LIN {X 0,Y 29.595,Z 545.275,A -85,B 0,C 180,E1 -30358.352,E2 -30358.352} C_VEL
LIN {X 0,Y 37.281,Z 542.804,A -85,B 0,C 180,E1 -30378.939,E2 -30378.939} C_VEL
LIN {X 0,Y 45.185,Z 539.847,A -85,B 0,C 180,E1 -30388.806,E2 -30388.806} C_VEL
LIN {X 0,Y 53.99,Z 535.853,A -85,B 0,C 180,E1 -30395.667,E2 -30395.667} C_VEL
LIN {X 0,Y 63.603,Z 530.542,A -85,B 0,C 180,E1 -30400.777,E2 -30400.777} C_VEL
LIN {X 0,Y 68.114,Z 527.764,A -85,B 0,C 180,E1 -30402.626,E2 -30402.626} C_VEL
LIN {X 0,Y 69.579,Z 526.593,A -85,B 0,C 180,E1 -30403.646,E2 -30403.646} C_VEL
LIN {X 0,Y 71.55,Z 524.834,A -85,B 0,C 180,E1 -30405.785,E2 -30405.785} C_VEL
LIN {X 0,Y 72.682,Z 523.453,A -85,B 0,C 180,E1 -30408.846,E2 -30408.846} C_VEL
LIN {X 0,Y 73.708,Z 521.841,A -85,B 0,C 180,E1 -30414.526,E2 -30414.526} C_VEL
LIN {X 0,Y 74.494,Z 520.765,A -85,B 0,C 180,E1 -30419.997,E2 -30419.997} C_VEL
LIN {X 0,Y 73.406,Z 521.71,A -85,B 0,C 180,E1 -30426.874,E2 -30426.874} C_VEL
LIN {X 0,Y 72.504,Z 523.18,A -85,B 0,C 180,E1 -30434.237,E2 -30434.237} C_VEL
LIN {X 0,Y 72.199,Z 523.884,A -85,B 0,C 180,E1 -30436.976,E2 -30436.976} C_VEL
LIN {X 0,Y 70.741,Z 526.379,A -85,B 0,C 180,E1 -30443.412,E2 -30443.412} C_VEL
LIN {X 0,Y 69.633,Z 527.972,A -85,B 0,C 180,E1 -30447.263,E2 -30447.263} C_VEL
LIN {X 0,Y 67.359,Z 530.893,A -85,B 0,C 180,E1 -30453.419,E2 -30453.419} C_VEL
LIN {X 0,Y 63.449,Z 535.475,A -85,B 0,C 180,E1 -30464.224,E2 -30464.224} C_VEL
LIN {X 0,Y 61.857,Z 538.776,A -85,B 0,C 180,E1 -30475.385,E2 -30475.385} C_VEL
LIN {X 0,Y 62.441,Z 540.641,A -85,B 0,C 180,E1 -30484.207,E2 -30484.207} C_VEL
LIN {X 0,Y 67.081,Z 542.547,A -85,B 0,C 180,E1 -30497.906,E2 -30497.906} C_VEL
LIN {X 0,Y 71.274,Z 542.971,A -85,B 0,C 180,E1 -30504.342,E2 -30504.342} C_VEL
LIN {X 0,Y 76.407,Z 542.961,A -85,B 0,C 180,E1 -30510.001,E2 -30510.001} C_VEL
LIN {X 0,Y 70.708,Z 542.926,A -85,B 0,C 180,E1 -30516.34,E2 -30516.34} C_VEL
LIN {X 0,Y 65.558,Z 542.209,A -85,B 0,C 180,E1 -30525.255,E2 -30525.255} C_VEL
LIN {X 0,Y 62.285,Z 540.421,A -85,B 0,C 180,E1 -30536.831,E2 -30536.831} C_VEL
LIN {X 0,Y 61.937,Z 538.036,A -85,B 0,C 180,E1 -30547.417,E2 -30547.417} C_VEL
LIN {X 0,Y 64.403,Z 534.161,A -85,B 0,C 180,E1 -30559.104,E2 -30559.104} C_VEL
LIN {X 0,Y 67.352,Z 530.892,A -85,B 0,C 180,E1 -30566.594,E2 -30566.594} C_VEL
LIN {X 0,Y 69.62,Z 527.97,A -85,B 0,C 180,E1 -30572.767,E2 -30572.767} C_VEL
LIN {X 0,Y 70.694,Z 526.411,A -85,B 0,C 180,E1 -30576.572,E2 -30576.572} C_VEL
LIN {X 0,Y 72.192,Z 523.889,A -85,B 0,C 180,E1 -30583.022,E2 -30583.022} C_VEL
LIN {X 0,Y 72.928,Z 522.452,A -85,B 0,C 180,E1 -30588.89,E2 -30588.89} C_VEL
LIN {X 0,Y 73.661,Z 521.458,A -85,B 0,C 180,E1 -30594.528,E2 -30594.528} C_VEL
LIN {X 0,Y 74.463,Z 520.789,A -85,B 0,C 180,E1 -30600.003,E2 -30600.003} C_VEL
LIN {X 0,Y 73.535,Z 522.043,A -85,B 0,C 180,E1 -30606.153,E2 -30606.153} C_VEL
LIN {X 0,Y 72.336,Z 523.174,A -85,B 0,C 180,E1 -30608.285,E2 -30608.285} C_VEL
LIN {X 0,Y 69.882,Z 525.092,A -85,B 0,C 180,E1 -30610.206,E2 -30610.206} C_VEL
LIN {X 0,Y 67.39,Z 526.857,A -85,B 0,C 180,E1 -30611.352,E2 -30611.352} C_VEL
LIN {X 0,Y 57.594,Z 532.628,A -85,B 0,C 180,E1 -30614.394,E2 -30614.394} C_VEL
LIN {X 0,Y 48.232,Z 537.171,A -85,B 0,C 180,E1 -30618.71,E2 -30618.71} C_VEL
LIN {X 0,Y 38.881,Z 540.786,A -85,B 0,C 180,E1 -30625.336,E2 -30625.336} C_VEL
LIN {X 0,Y 33.037,Z 542.591,A -85,B 0,C 180,E1 -30631.685,E2 -30631.685} C_VEL
LIN {X 0,Y 23.563,Z 545.062,A -85,B 0,C 180,E1 -30653.374,E2 -30653.374} C_VEL
LIN {X 0,Y 20.769,Z 545.664,A -85,B 0,C 180,E1 -30670.217,E2 -30670.217} C_VEL
LIN {X 0,Y 20.025,Z 545.83,A -85,B 0,C 180,E1 -30689.996,E2 -30689.996} C_VEL
LIN {X 0,Y 20.768,Z 545.664,A -85,B 0,C 180,E1 -30709.775,E2 -30709.775} C_VEL
LIN {X 0,Y 23.561,Z 545.062,A -85,B 0,C 180,E1 -30726.62,E2 -30726.62} C_VEL
LIN {X 0,Y 33.035,Z 542.592,A -85,B 0,C 180,E1 -30748.313,E2 -30748.313} C_VEL
LIN {X 0,Y 41.939,Z 539.635,A -85,B 0,C 180,E1 -30757.165,E2 -30757.165} C_VEL
LIN {X 0,Y 51.468,Z 535.641,A -85,B 0,C 180,E1 -30762.905,E2 -30762.905} C_VEL
LIN {X 0,Y 61.319,Z 530.507,A -85,B 0,C 180,E1 -30766.938,E2 -30766.938} C_VEL
LIN {X 0,Y 64.658,Z 528.588,A -85,B 0,C 180,E1 -30768.017,E2 -30768.017} C_VEL
LIN {X 0,Y 66.911,Z 526.732,A -85,B 0,C 180,E1 -30771.207,E2 -30771.207} C_VEL
LIN {X 0,Y 67.428,Z 526.025,A -85,B 0,C 180,E1 -30774.014,E2 -30774.014} C_VEL
LIN {X 0,Y 68.512,Z 524.866,A -85,B 0,C 180,E1 -30779.997,E2 -30779.997} C_VEL
LIN {X 0,Y 67.504,Z 525.562,A -85,B 0,C 180,E1 -30786.094,E2 -30786.094} C_VEL
LIN {X 0,Y 66.682,Z 526.625,A -85,B 0,C 180,E1 -30792.165,E2 -30792.165} C_VEL
LIN {X 0,Y 65.975,Z 527.63,A -85,B 0,C 180,E1 -30796.526,E2 -30796.526} C_VEL
LIN {X 0,Y 64.335,Z 529.517,A -85,B 0,C 180,E1 -30802.475,E2 -30802.475} C_VEL
LIN {X 0,Y 62.896,Z 531.158,A -85,B 0,C 180,E1 -30806.635,E2 -30806.635} C_VEL
LIN {X 0,Y 61.261,Z 532.718,A -85,B 0,C 180,E1 -30810.64,E2 -30810.64} C_VEL
LIN {X 0,Y 56.854,Z 536.807,A -85,B 0,C 180,E1 -30822.128,E2 -30822.128} C_VEL
LIN {X 0,Y 55.221,Z 539.024,A -85,B 0,C 180,E1 -30830.482,E2 -30830.482} C_VEL
LIN {X 0,Y 55.213,Z 541.318,A -85,B 0,C 180,E1 -30842.993,E2 -30842.993} C_VEL
LIN {X 0,Y 58.568,Z 542.807,A -85,B 0,C 180,E1 -30856.116,E2 -30856.116} C_VEL
LIN {X 0,Y 63.481,Z 543.319,A -85,B 0,C 180,E1 -30865.084,E2 -30865.084} C_VEL
LIN {X 0,Y 67.405,Z 543.228,A -85,B 0,C 180,E1 -30870.001,E2 -30870.001} C_VEL
LIN {X 0,Y 62.439,Z 543.236,A -85,B 0,C 180,E1 -30876.464,E2 -30876.464} C_VEL
LIN {X 0,Y 58.183,Z 542.744,A -85,B 0,C 180,E1 -30884.925,E2 -30884.925} C_VEL
LIN {X 0,Y 54.911,Z 540.671,A -85,B 0,C 180,E1 -30900.796,E2 -30900.796} C_VEL
LIN {X 0,Y 55.817,Z 537.952,A -85,B 0,C 180,E1 -30913.825,E2 -30913.825} C_VEL
LIN {X 0,Y 59.648,Z 534.186,A -85,B 0,C 180,E1 -30925.566,E2 -30925.566} C_VEL
LIN {X 0,Y 61.25,Z 532.717,A -85,B 0,C 180,E1 -30929.382,E2 -30929.382} C_VEL
LIN {X 0,Y 62.895,Z 531.138,A -85,B 0,C 180,E1 -30933.455,E2 -30933.455} C_VEL
LIN {X 0,Y 64.302,Z 529.536,A -85,B 0,C 180,E1 -30937.513,E2 -30937.513} C_VEL
LIN {X 0,Y 65.967,Z 527.63,A -85,B 0,C 180,E1 -30943.508,E2 -30943.508} C_VEL
LIN {X 0,Y 66.69,Z 526.619,A -85,B 0,C 180,E1 -30947.836,E2 -30947.836} C_VEL
LIN {X 0,Y 67.533,Z 525.536,A -85,B 0,C 180,E1 -30954.03,E2 -30954.03} C_VEL
LIN {X 0,Y 68.475,Z 524.89,A -85,B 0,C 180,E1 -30960.003,E2 -30960.003} C_VEL
LIN {X 0,Y 67.404,Z 526.04,A -85,B 0,C 180,E1 -30965.988,E2 -30965.988} C_VEL
LIN {X 0,Y 66.816,Z 526.795,A -85,B 0,C 180,E1 -30968.807,E2 -30968.807} C_VEL
LIN {X 0,Y 64.662,Z 528.587,A -85,B 0,C 180,E1 -30971.986,E2 -30971.986} C_VEL
LIN {X 0,Y 57.594,Z 532.628,A -85,B 0,C 180,E1 -30974.394,E2 -30974.394} C_VEL
LIN {X 0,Y 52.388,Z 535.105,A -85,B 0,C 180,E1 -30975.853,E2 -30975.853} C_VEL
LIN {X 0,Y 46.882,Z 537.38,A -85,B 0,C 180,E1 -30976.499,E2 -30976.499} C_VEL
LIN {X 0,Y 35.537,Z 540.932,A -85,B 0,C 180,E1 -30977.575,E2 -30977.575} C_VEL
LIN {X 0,Y 29.088,Z 542.618,A -85,B 0,C 180,E1 -30980.837,E2 -30980.837} C_VEL
LIN {X 0,Y 28.223,Z 542.755,A -85,B 0,C 180,E1 -30981.7,E2 -30981.7} C_VEL
LIN {X 0,Y 18.344,Z 544.85,A -85,B 0,C 180,E1 -30999.978,E2 -30999.978} C_VEL
LIN {X 0,Y 14.273,Z 545.452,A -85,B 0,C 180,E1 -31020.494,E2 -31020.494} C_VEL
LIN {X 0,Y 12.932,Z 545.619,A -85,B 0,C 180,E1 -31049.993,E2 -31049.993} C_VEL
LIN {X 0,Y 14.271,Z 545.452,A -85,B 0,C 180,E1 -31079.495,E2 -31079.495} C_VEL
LIN {X 0,Y 18.342,Z 544.85,A -85,B 0,C 180,E1 -31100.016,E2 -31100.016} C_VEL
LIN {X 0,Y 29.909,Z 542.38,A -85,B 0,C 180,E1 -31120.024,E2 -31120.024} C_VEL
LIN {X 0,Y 39.72,Z 539.422,A -85,B 0,C 180,E1 -31126.685,E2 -31126.685} C_VEL
LIN {X 0,Y 49.842,Z 535.429,A -85,B 0,C 180,E1 -31130.75,E2 -31130.75} C_VEL
LIN {X 0,Y 60.111,Z 530.295,A -85,B 0,C 180,E1 -31133.565,E2 -31133.565} C_VEL
LIN {X 0,Y 61.605,Z 529.239,A -85,B 0,C 180,E1 -31136.726,E2 -31136.726} C_VEL
LIN {X 0,Y 62.267,Z 528.721,A -85,B 0,C 180,E1 -31139.996,E2 -31139.996} C_VEL
LIN {X 0,Y 61.158,Z 529.332,A -85,B 0,C 180,E1 -31146.595,E2 -31146.595} C_VEL
LIN {X 0,Y 60.017,Z 530.426,A -85,B 0,C 180,E1 -31153.541,E2 -31153.541} C_VEL
LIN {X 0,Y 58.992,Z 531.466,A -85,B 0,C 180,E1 -31157.629,E2 -31157.629} C_VEL
LIN {X 0,Y 57.693,Z 532.582,A -85,B 0,C 180,E1 -31161.431,E2 -31161.431} C_VEL
LIN {X 0,Y 55.312,Z 534.438,A -85,B 0,C 180,E1 -31167.203,E2 -31167.203} C_VEL
LIN {X 0,Y 51.732,Z 537.05,A -85,B 0,C 180,E1 -31175.405,E2 -31175.405} C_VEL
LIN {X 0,Y 48.796,Z 539.572,A -85,B 0,C 180,E1 -31186.059,E2 -31186.059} C_VEL
LIN {X 0,Y 48.243,Z 542.159,A -85,B 0,C 180,E1 -31204.087,E2 -31204.087} C_VEL
LIN {X 0,Y 50.802,Z 543.149,A -85,B 0,C 180,E1 -31215.538,E2 -31215.538} C_VEL
LIN {X 0,Y 56.3,Z 543.561,A -85,B 0,C 180,E1 -31226.94,E2 -31226.94} C_VEL
LIN {X 0,Y 58.461,Z 543.495,A -85,B 0,C 180,E1 -31230.001,E2 -31230.001} C_VEL
LIN {X 0,Y 53.721,Z 543.497,A -85,B 0,C 180,E1 -31237.519,E2 -31237.519} C_VEL
LIN {X 0,Y 50.276,Z 543.063,A -85,B 0,C 180,E1 -31246.237,E2 -31246.237} C_VEL
LIN {X 0,Y 48.02,Z 541.878,A -85,B 0,C 180,E1 -31258.592,E2 -31258.592} C_VEL
LIN {X 0,Y 49.079,Z 539.271,A -85,B 0,C 180,E1 -31275.726,E2 -31275.726} C_VEL
LIN {X 0,Y 53.19,Z 536.073,A -85,B 0,C 180,E1 -31288.099,E2 -31288.099} C_VEL
LIN {X 0,Y 55.302,Z 534.438,A -85,B 0,C 180,E1 -31292.823,E2 -31292.823} C_VEL
LIN {X 0,Y 57.64,Z 532.607,A -85,B 0,C 180,E1 -31298.548,E2 -31298.548} C_VEL
LIN {X 0,Y 58.984,Z 531.465,A -85,B 0,C 180,E1 -31302.407,E2 -31302.407} C_VEL
LIN {X 0,Y 60.014,Z 530.428,A -85,B 0,C 180,E1 -31306.459,E2 -31306.459} C_VEL
LIN {X 0,Y 61.163,Z 529.33,A -85,B 0,C 180,E1 -31313.406,E2 -31313.406} C_VEL
LIN {X 0,Y 62.253,Z 528.729,A -85,B 0,C 180,E1 -31320.004,E2 -31320.004} C_VEL
LIN {X 0,Y 61.578,Z 529.254,A -85,B 0,C 180,E1 -31323.275,E2 -31323.275} C_VEL
LIN {X 0,Y 60.113,Z 530.294,A -85,B 0,C 180,E1 -31326.429,E2 -31326.429} C_VEL
LIN {X 0,Y 49.845,Z 535.428,A -85,B 0,C 180,E1 -31329.253,E2 -31329.253} C_VEL
LIN {X 0,Y 39.723,Z 539.421,A -85,B 0,C 180,E1 -31333.316,E2 -31333.316} C_VEL
LIN {X 0,Y 29.912,Z 542.379,A -85,B 0,C 180,E1 -31339.974,E2 -31339.974} C_VEL
LIN {X 0,Y 28.223,Z 542.755,A -85,B 0,C 180,E1 -31341.7,E2 -31341.7} C_VEL
LIN {X 0,Y 22.938,Z 543.892,A -85,B 0,C 180,E1 -31347.166,E2 -31347.166} C_VEL
LIN {X 0,Y 17.452,Z 544.74,A -85,B 0,C 180,E1 -31353.279,E2 -31353.279} C_VEL
LIN {X 0,Y 7.362,Z 545.435,A -85,B 0,C 180,E1 -31386.239,E2 -31386.239} C_VEL
LIN {X 0,Y 7.357,Z 545.291,A -85,B 0,C 180,E1 -31452.017,E2 -31452.017} C_VEL
LIN {X 0,Y 14.81,Z 544.638,A -85,B 0,C 180,E1 -31481.617,E2 -31481.617} C_VEL
LIN {X 0,Y 28.279,Z 542.167,A -85,B 0,C 180,E1 -31493.727,E2 -31493.727} C_VEL
LIN {X 0,Y 38.705,Z 539.21,A -85,B 0,C 180,E1 -31497.007,E2 -31497.007} C_VEL
LIN {X 0,Y 49.201,Z 535.216,A -85,B 0,C 180,E1 -31498.992,E2 -31498.992} C_VEL
LIN {X 0,Y 55.815,Z 532.215,A -85,B 0,C 180,E1 -31499.996,E2 -31499.996} C_VEL
LIN {X 0,Y 54.509,Z 532.847,A -85,B 0,C 180,E1 -31507.404,E2 -31507.404} C_VEL
LIN {X 0,Y 52.661,Z 534.088,A -85,B 0,C 180,E1 -31515.476,E2 -31515.476} C_VEL
LIN {X 0,Y 51.739,Z 534.714,A -85,B 0,C 180,E1 -31518.047,E2 -31518.047} C_VEL
LIN {X 0,Y 49.656,Z 536.09,A -85,B 0,C 180,E1 -31522.702,E2 -31522.702} C_VEL
LIN {X 0,Y 43.786,Z 539.514,A -85,B 0,C 180,E1 -31536.631,E2 -31536.631} C_VEL
LIN {X 0,Y 41.503,Z 541.167,A -85,B 0,C 180,E1 -31547.367,E2 -31547.367} C_VEL
LIN {X 0,Y 42.116,Z 543.318,A -85,B 0,C 180,E1 -31570.506,E2 -31570.506} C_VEL
LIN {X 0,Y 45.091,Z 543.757,A -85,B 0,C 180,E1 -31581.035,E2 -31581.035} C_VEL
LIN {X 0,Y 49.616,Z 543.758,A -85,B 0,C 180,E1 -31590.002,E2 -31590.002} C_VEL
LIN {X 0,Y 43.443,Z 543.542,A -85,B 0,C 180,E1 -31603.936,E2 -31603.936} C_VEL
LIN {X 0,Y 40.872,Z 542.408,A -85,B 0,C 180,E1 -31621.057,E2 -31621.057} C_VEL
LIN {X 0,Y 42.45,Z 540.3,A -85,B 0,C 180,E1 -31638.536,E2 -31638.536} C_VEL
LIN {X 0,Y 48.026,Z 536.976,A -85,B 0,C 180,E1 -31653.965,E2 -31653.965} C_VEL
LIN {X 0,Y 49.641,Z 536.094,A -85,B 0,C 180,E1 -31657.316,E2 -31657.316} C_VEL
LIN {X 0,Y 51.71,Z 534.715,A -85,B 0,C 180,E1 -31662.064,E2 -31662.064} C_VEL
LIN {X 0,Y 52.615,Z 534.109,A -85,B 0,C 180,E1 -31664.51,E2 -31664.51} C_VEL
LIN {X 0,Y 54.511,Z 532.845,A -85,B 0,C 180,E1 -31672.597,E2 -31672.597} C_VEL
LIN {X 0,Y 55.806,Z 532.22,A -85,B 0,C 180,E1 -31680.004,E2 -31680.004} C_VEL
LIN {X 0,Y 45.7,Z 536.747,A -85,B 0,C 180,E1 -31681.554,E2 -31681.554} C_VEL
LIN {X 0,Y 35.222,Z 540.362,A -85,B 0,C 180,E1 -31683.893,E2 -31683.893} C_VEL
LIN {X 0,Y 25.646,Z 542.703,A -85,B 0,C 180,E1 -31687.603,E2 -31687.603} C_VEL
LIN {X 0,Y 14.813,Z 544.638,A -85,B 0,C 180,E1 -31698.38,E2 -31698.38} C_VEL
LIN {X 0,Y 8.81,Z 545.24,A -85,B 0,C 180,E1 -31717.075,E2 -31717.075} C_VEL
LIN {X 0,Y 5.826,Z 545.408,A -85,B 0,C 180,E1 -31769.985,E2 -31769.985} C_VEL
LIN {X 0,Y 7.357,Z 545.291,A -85,B 0,C 180,E1 -31812.017,E2 -31812.017} C_VEL
LIN {X 0,Y 10.044,Z 545.109,A -85,B 0,C 180,E1 -31831.192,E2 -31831.192} C_VEL
LIN {X 0,Y 16.341,Z 544.329,A -85,B 0,C 180,E1 -31852.358,E2 -31852.358} C_VEL
LIN {X 0,Y 27.025,Z 542.304,A -85,B 0,C 180,E1 -31865.805,E2 -31865.805} C_VEL
LIN {X 0,Y 32.715,Z 540.862,A -85,B 0,C 180,E1 -31867.68,E2 -31867.68} C_VEL
LIN {X 0,Y 34.634,Z 540.361,A -85,B 0,C 180,E1 -31867.71,E2 -31867.71} C_VEL
LIN {X 0,Y 42.529,Z 537.777,A -85,B 0,C 180,E1 -31867.489,E2 -31867.489} C_VEL
LIN {X 0,Y 47.334,Z 536.029,A -85,B 0,C 180,E1 -31868.534,E2 -31868.534} C_VEL
LIN {X 0,Y 44.177,Z 537.55,A -85,B 0,C 180,E1 -31877.355,E2 -31877.355} C_VEL
LIN {X 0,Y 39.462,Z 539.757,A -85,B 0,C 180,E1 -31887.073,E2 -31887.073} C_VEL
LIN {X 0,Y 35.838,Z 541.414,A -85,B 0,C 180,E1 -31898.338,E2 -31898.338} C_VEL
LIN {X 0,Y 34.257,Z 543.57,A -85,B 0,C 180,E1 -31925.779,E2 -31925.779} C_VEL
LIN {X 0,Y 36.638,Z 544.012,A -85,B 0,C 180,E1 -31938.943,E2 -31938.943} C_VEL
LIN {X 0,Y 40.886,Z 544.018,A -85,B 0,C 180,E1 -31950.002,E2 -31950.002} C_VEL
LIN {X 0,Y 36.079,Z 543.94,A -85,B 0,C 180,E1 -31963.127,E2 -31963.127} C_VEL
LIN {X 0,Y 33.821,Z 542.994,A -85,B 0,C 180,E1 -31983.789,E2 -31983.789} C_VEL
LIN {X 0,Y 36.567,Z 540.999,A -85,B 0,C 180,E1 -32004.797,E2 -32004.797} C_VEL
LIN {X 0,Y 39.444,Z 539.758,A -85,B 0,C 180,E1 -32012.989,E2 -32012.989} C_VEL
LIN {X 0,Y 44.168,Z 537.55,A -85,B 0,C 180,E1 -32022.697,E2 -32022.697} C_VEL
LIN {X 0,Y 47.3,Z 536.044,A -85,B 0,C 180,E1 -32031.46,E2 -32031.46} C_VEL
LIN {X 0,Y 42.531,Z 537.776,A -85,B 0,C 180,E1 -32032.514,E2 -32032.514} C_VEL
LIN {X 0,Y 35.457,Z 540.15,A -85,B 0,C 180,E1 -32032.34,E2 -32032.34} C_VEL
LIN {X 0,Y 28.401,Z 541.955,A -85,B 0,C 180,E1 -32031.84,E2 -32031.84} C_VEL
LIN {X 0,Y 14.27,Z 544.426,A -85,B 0,C 180,E1 -32030.088,E2 -32030.088} C_VEL
LIN {X 0,Y 7.253,Z 545.029,A -85,B 0,C 180,E1 -32025.723,E2 -32025.723} C_VEL
LIN {X 0,Y 1.286,Z 545.196,A -85,B 0,C 180,E1 -31950.068,E2 -31950.068} C_VEL
LIN {X 0,Y 7.25,Z 545.029,A -85,B 0,C 180,E1 -31874.283,E2 -31874.283} C_VEL
LIN {X 0,Y 14.267,Z 544.426,A -85,B 0,C 180,E1 -31869.914,E2 -31869.914} C_VEL
LIN {X 0,Y 28.398,Z 541.955,A -85,B 0,C 180,E1 -31868.162,E2 -31868.162} C_VEL
LIN {X 0,Y 34.634,Z 540.361,A -85,B 0,C 180,E1 -31867.71,E2 -31867.71} C_VEL
LIN {X 0,Y 35.253,Z 540.211,A -85,B 0,C 180,E1 -31868.775,E2 -31868.775} C_VEL
LIN {X 0,Y 35.21,Z 540.264,A -85,B 0,C 180,E1 -31872.001,E2 -31872.001} C_VEL
LIN {X 0,Y 33.985,Z 540.688,A -85,B 0,C 180,E1 -31877.327,E2 -31877.327} C_VEL
LIN {X 0,Y 29.844,Z 542.226,A -85,B 0,C 180,E1 -31890.972,E2 -31890.972} C_VEL
LIN {X 0,Y 27.416,Z 543.169,A -85,B 0,C 180,E1 -31905.259,E2 -31905.259} C_VEL
LIN {X 0,Y 28.304,Z 544.266,A -85,B 0,C 180,E1 -31935.626,E2 -31935.626} C_VEL
LIN {X 0,Y 32.248,Z 544.275,A -85,B 0,C 180,E1 -31950.003,E2 -31950.003} C_VEL
LIN {X 0,Y 28.306,Z 544.266,A -85,B 0,C 180,E1 -31964.379,E2 -31964.379} C_VEL
LIN {X 0,Y 26.882,Z 543.558,A -85,B 0,C 180,E1 -31988.355,E2 -31988.355} C_VEL
LIN {X 0,Y 32.945,Z 541.106,A -85,B 0,C 180,E1 -32017.598,E2 -32017.598} C_VEL
LIN {X 0,Y 30.242,Z 541.743,A -85,B 0,C 180,E1 -32018.371,E2 -32018.371} C_VEL
LIN {X 0,Y 17.023,Z 544.213,A -85,B 0,C 180,E1 -32005.666,E2 -32005.666} C_VEL
LIN {X 0,Y 11.353,Z 544.817,A -85,B 0,C 180,E1 -31988.255,E2 -31988.255} C_VEL
LIN {X 0,Y 8.384,Z 544.985,A -85,B 0,C 180,E1 -31950.01,E2 -31950.01} C_VEL
LIN {X 0,Y 11.351,Z 544.817,A -85,B 0,C 180,E1 -31911.757,E2 -31911.757} C_VEL
LIN {X 0,Y 17.021,Z 544.214,A -85,B 0,C 180,E1 -31894.34,E2 -31894.34} C_VEL
LIN {X 0,Y 30.24,Z 541.744,A -85,B 0,C 180,E1 -31881.632,E2 -31881.632} C_VEL
LIN {X 0,Y 32.979,Z 541.099,A -85,B 0,C 180,E1 -31882.44,E2 -31882.44} C_VEL
LIN {X 0,Y 27.416,Z 543.169,A -85,B 0,C 180,E1 -31905.259,E2 -31905.259} C_VEL
LIN {X 0,Y 26.068,Z 543.59,A -85,B 0,C 180,E1 -31910.071,E2 -31910.071} C_VEL
LIN {X 0,Y 20.556,Z 544.355,A -85,B 0,C 180,E1 -31922.928,E2 -31922.928} C_VEL
LIN {X 0,Y 20.177,Z 544.509,A -85,B 0,C 180,E1 -31929.171,E2 -31929.171} C_VEL
LIN {X 0,Y 23.622,Z 544.531,A -85,B 0,C 180,E1 -31950.004,E2 -31950.004} C_VEL
LIN {X 0,Y 19.788,Z 544.377,A -85,B 0,C 180,E1 -31977.889,E2 -31977.889} C_VEL
LIN {X 0,Y 17.506,Z 544.605,A -85,B 0,C 180,E1 -31973.675,E2 -31973.675} C_VEL
LIN {X 0,Y 15.473,Z 544.774,A -85,B 0,C 180,E1 -31950.006,E2 -31950.006} C_VEL
LIN {X 0,Y 17.504,Z 544.605,A -85,B 0,C 180,E1 -31926.334,E2 -31926.334} C_VEL
LIN {X 0,Y 19.795,Z 544.376,A -85,B 0,C 180,E1 -31922.094,E2 -31922.094} C_VEL
LIN {X 0,Y 20.177,Z 544.509,A -85,B 0,C 180,E1 -31929.171,E2 -31929.171} C_VEL
LIN {X 0,Y 20.663,Z 546.506,A -85,B 0,C 180,E1 -31934.308,E2 -31934.308} C_VEL
LIN {X 0,Y 20.663,Z 600,A -85,B 0,C 180,E1 -31934.308,E2 -31934.308} C_VEL
LIN {X 0,Y 20.663,Z 600,A -85,B 0,C 180,E1 -31934.308,E2 -31934.308}

QRS_NEXT_CUT()

QRS_NEXT()
QRS_HOME()

END
